FUNCTION_BLOCK FB_EstopLED
VAR_INPUT
	bEstopSignal : BOOL;
	bSafetySystemSignal : BOOL;
END_VAR
VAR_OUTPUT
	bLEDOutput : BOOL;
END_VAR
VAR
	tOnBlinkTime : TIME;
	nNumOfOnBlinks : INT;
	tLEDOffTime : TIME;
	fbLEDPulse: FB_Pulse;
	fbBlinkPulse: FB_Pulse;
	bBlinkEn: BOOL;
	tTotalTimeOn: TIME;
	tOffBlinkTime: TIME;
END_VAR

IF NOT bEstopSignal THEN
	tOnBlinkTime := T#250MS;
	tOffBlinkTime := T#250MS;
	nNumOfOnBlinks := 3;
	tLEDOffTime := T#1000MS;
	bBlinkEn := TRUE;
	bLEDOutput := fbBlinkPulse.bPulse;	
ELSIF NOT bSafetySystemSignal THEN
	tOnBlinkTime := T#1000MS;
	tOffBlinkTime := T#250MS;
	nNumOfOnBlinks := 1;
	tLEDOffTime := T#1000MS;
	bBlinkEn := TRUE;
	bLEDOutput := fbBlinkPulse.bPulse;	
ELSE
	bLEDOutput := TRUE;	
	bBlinkEn := FALSE;
END_IF

tTotalTimeOn := DINT_TO_TIME((TIME_TO_DINT(tOnBlinkTime) * (nNumOfOnBlinks)) + (TIME_TO_DINT(tOffBlinkTime) * (nNumOfOnBlinks - 1)));
fbLEDPulse(bEnable:= bBlinkEn, tTimeOn:= tTotalTimeOn, tTimeOff:= tLEDOffTime, bPulse=> );
fbBlinkPulse(bEnable:= fbLEDPulse.bPulse, tTimeOn:= tOnBlinkTime, tTimeOff:= tOffBlinkTime, bPulse=> );

END_FUNCTION_BLOCK

(* stored: Version 1.1.0.1, ProductVersion 3.1.4022.3
   POU FB_EstopLED: Id {1db509ae-796c-47b6-b418-89bcbd0efe14}, SpecialFunc None *)
